PROGRAM EM04_Follower3
VAR
	ref_Master: REFERENCE TO UDT_AXISADMIN;
	ref_Follower: REFERENCE TO UDT_AXISADMIN;
	Ref_MachineStateModel: REFERENCE TO PackMlv3_StateModel;
	Ref_Unit: REFERENCE TO UDT_UnitAdmin;
	EM_No: INT:=4;
	tonAbortingWatchDog: TON;
	tonStoppingWatchDog: Ton;
	MC_CamIn_Follower: MC_CamIn;

	MC_CamTableSelect_Follower: MC_CamTableSelect;
	CamTableFollower: MC_CAM_REF;
	table1: ARRAY[1..2] OF MC_MotionFunctionPoint; (*用于定义电子凸轮表中的关键点*)


    MC_ReadCamTableSlaveDynamicsFollwer: MC_ReadCamTableSlaveDynamics;
	
	tonFollowerSeq: TON;
	FollowerSeq: SequenceTransfer;	
	
	i: INT;
	lrPosCnt: INT;
	bRecipeComplete: BOOL;
	bBeltInRange: BOOL;
	iLastSeq: INT;
END_VAR

VAR CONSTANT
	iCamID: MC_CAM_ID:=3;		
END_VAR

(*减速比10/1 同步轮周长400 ，皮带总长11600，58个工位，工位间距200
28个工位后开始落料*)
Ref_MachineStateModel REF= UN01_MachineStateModel;
Ref_Unit REF=Unit01;
ref_Master REF= arVirtualAxisAdmin[1];
ref_Follower REF= arRealAxisAdmin[43];
MainRoution();
CM01_Cam();
SR999_Faulthandler();

ACTION CM01_Cam:
//凸轮1曲线
camTableFollower.ArraySize:=SIZEOF(table1);
camTableFollower.NoOfColumns:=1;
camTableFollower.NoOfRows:=2;
camTableFollower.pArray:=ADR(table1);
camTableFollower.TableType:=MC_TABLETYPE_MOTIONFUNCTION;

table1[1].FunctionType:=MOTIONFUNCTYPE_POLYNOM1;
table1[1].MasterPos:=0;
table1[1].SlavePos:=0;
table1[1].PointIndex:=1;
table1[1].PointType:=MOTIONPOINTTYPE_MOTION;
		
table1[2].FunctionType:=MOTIONFUNCTYPE_POLYNOM1;
table1[2].MasterPos:=200;
table1[2].SlavePos:=200;
table1[2].PointIndex:=2;
table1[2].PointType:=MOTIONPOINTTYPE_MOTION;

MC_CamIn_Follower(
	Master:= ref_Master.Axis, 
	Slave:= ref_Follower.Axis, 
	Execute:= ref_Follower.i.CamIn , 
	MasterOffset:= , 
	SlaveOffset:= , 
	MasterScaling:= 1, 
	SlaveScaling:= 1, 
	StartMode:= MC_STARTMODE_ABSOLUTE, 
	CamTableID:= iCamID, 
	BufferMode:= , 
	Options:= , 
	InSync=> , 
	Busy=> , 
	Active=> , 
	CommandAborted=> , 
	Error=> , 
	ErrorID=> );
	
MC_CamTableSelect_Follower(
	Master:= ref_Master.Axis, 
	Slave:= ref_Follower.Axis, 
	CamTable:= CamTableFollower, 
	Execute:= ref_Follower.i.SelectCamTable , 
	Periodic:= TRUE, 
	MasterAbsolute:= , 
	SlaveAbsolute:= , 
	CamTableID:= iCamID, 
	Done=> ref_Follower.o.SelectCamTableDone, 
	Busy=> , 
	Error=> , 
	ErrorID=> );	
	
MC_ReadCamTableSlaveDynamicsFollwer(
	Execute:= , 
	CamTableID:=iCamID , 
	MasterPosition:=ref_Master.o.ActPos, 
	Done=> , 
	Busy=> , 
	Error=> , 
	ErrorID=> , 
	SlavePosition=> , 
	SlaveVelocity=> , 
	SlaveAcceleration=> );
END_ACTION

ACTION CM02_Follower:
CASE FollowerSeq.Now OF
	0: 	   
	   IF Ref_MachineStateModel.Sts_Resetting  THEN
          FollowerSeq(ExeCute:=TRUE , Next:= Seq_Resetting);  
	   END_IF	
	
	   IF Ref_MachineStateModel.Sts_Stopping  THEN
		  FollowerSeq(ExeCute:=TRUE , Next:= Seq_Stopping);   
	   END_IF
	   IF Ref_MachineStateModel.Sts_Execute  THEN
		  FollowerSeq(ExeCute:= TRUE, Next:= 110);   
	   END_IF	   
{#region resetting}	   
	Seq_Resetting:
		IF NOT ref_Follower.o.PowerOn  THEN;
		   ref_Follower.i.Enable:=TRUE;
		ELSE
		   FollowerSeq(ExeCute:=TRUE , Next:= 20); 
		END_IF
	    IF Ref_MachineStateModel.Sts_Stopping  THEN
		   FollowerSeq(ExeCute:= TRUE, Next:= Seq_Stopping);  
	    END_IF
		
	20:	
		IF NOT glb_AllAxisHomed_UN01 THEN
			FollowerSeq(ExeCute:=TRUE , Next:= 21);  
			ELSE
			FollowerSeq(ExeCute:=TRUE , Next:= 30); 
		END_IF
	   
	21:
	   iLastSeq:=0;
	   glb_lrBelt3TargetCnt:=0;
	   glb_lrBelt3WrkCnt:=0;
	   glb_lrBelt3ValidCnt:=0;
	   bRecipeComplete:=FALSE;
	   arDropBufferCyclinder[1].i.ActiveIn:=TRUE;
	   arDropBufferCyclinder[1].i.ActiveOut:=FALSE;
	   MEMSET(destAddr:= ADR(glb_BinBelt3), fillByte:= 0, n:= SIZEOF(glb_BinBelt3));      
	   FollowerSeq(ExeCute:=TRUE , Next:= 22); 
	22:
       tonFollowerSeq(IN:=TRUE , PT:=T#1S , Q=> , ET=> );
       IF tonFollowerSeq.Q AND arDropBufferCyclinder[1].I.InSensor 
       AND arDropBufferCyclinder[2].i.InSensor THEN
		   tonFollowerSeq(IN:=FALSE , PT:=T#1S , Q=> , ET=> );
		   FollowerSeq(ExeCute:=TRUE , Next:= 23); 
       END_IF 
	   
	23:
	   ref_Follower.i.Home:=TRUE;
	   IF ref_Follower.o.HomeDone THEN
		   ref_Follower.i.Home:=FALSE;
		   FollowerSeq(ExeCute:=TRUE , Next:= 24); 
	   ELSE IF Ref_MachineStateModel.Sts_Stopping  THEN
		       ref_Follower.i.Home:=FALSE;
			   ref_Follower.i.Stop:=TRUE;
               FollowerSeq(ExeCute:=TRUE , Next:= Seq_Stopping);   
	        END_IF	   
	   END_IF	
		
    24: 
		glb_BinBelt3.bin[1].arDrop[HMI_B3DropBinNo1]:=TRUE;
		glb_BinBelt3.bin[1].arDrop[HMI_B3DropBinNo2]:=TRUE;
		glb_BinBelt3.bin[1].arDrop[HMI_B3DropBinNo3]:=TRUE;
        lrPosCnt:=1;
		ref_Follower.i.Pos:=0;		
		FollowerSeq(ExeCute:=TRUE , Next:= 25);
		
	25:
        IF ref_Follower.o.StandStill THEN
		   FollowerSeq(Execute:= TRUE, Next:= 30);   
	    END_IF
		
    30:	//生产复位
	    ref_Follower.i.MoveAbs:=TRUE; 	
    	IF  ref_Follower.o.CmdDone THEN
		    ref_Follower.i.MoveAbs:=FALSE;
            FollowerSeq(Execute:= TRUE, Next:= Seq_ResettingDone);    	
		END_IF

		
   	Seq_ResettingDone: 
         IF NOT Ref_MachineStateModel.Sts_Resetting THEN
			FollowerSeq(ExeCute:=TRUE , Next:= 0); 	
		 END_IF	   
{end_region}
	
    //自动运行
    110:
        IF iLastSeq>100 THEN
	       FollowerSeq(ExeCute:=TRUE , Next:= iLastSeq);
        ELSE 
		   FollowerSeq(ExeCute:=TRUE , Next:= 111);
		END_IF
    111: 
        IF glb_BinBelt1.bin[HMI_B1DropBinNo].arDrop[HMI_B1DropBinNo] THEN //等待皮带1倒药
		   FollowerSeq(ExeCute:=TRUE , Next:= 112);
		END_IF
		
		IF NOT glb_BinBelt1.bin[HMI_B1DropBinNo].arDrop[HMI_B1DropBinNo] 
		   AND glb_lrBelt3ValidCnt > 0  THEN // AND glb_lrBelt1WrkCnt=0 
			FollowerSeq(ExeCute:=TRUE , Next:= 120);
		END_IF
		
		IF Ref_MachineStateModel.Sts_Stopping  THEN
			FollowerSeq(ExeCute:=TRUE , Next:= Seq_Stopping);   
		END_IF   		
    112:
		   glb_BinBelt3.bin[1].arDrop[HMI_B3DropBinNo1]:=TRUE;
//		   glb_BinBelt3.bin[1].arDrop[HMI_B3DropBinNo2]:=FALSE;
//		   glb_BinBelt3.bin[1].arDrop[HMI_B3DropBinNo3]:=FALSE; 
           FollowerSeq(ExeCute:=TRUE , Next:= 120); 	
    120:  
	      IF NOT glb_BinBelt3.bin[HMI_B3DropBinNo1].arDrop[HMI_B3DropBinNo1] 
          AND NOT glb_BinBelt3.bin[HMI_B3DropBinNo2].arDrop[HMI_B3DropBinNo2] THEN 
              FollowerSeq(ExeCute:=TRUE , Next:= 121); 	
		  END_IF
		  IF Ref_MachineStateModel.Sts_Stopping  THEN
		     FollowerSeq(ExeCute:=TRUE , Next:= Seq_Stopping);   
	      END_IF
		  
    121: 
         IF NOT glb_BinBelt3.bin[HMI_B3DropBinNo3].arDrop[HMI_B3DropBinNo3] THEN
             FollowerSeq(ExeCute:=TRUE , Next:= 130); 	
	     ELSE 
		     FollowerSeq(ExeCute:=TRUE , Next:= 200); //往皮带4倒药	
         END_IF
	130:  
	      ref_Follower.i.Pos:=ref_Follower.i.Pos+200;
	      FollowerSeq(ExeCute:=TRUE ,Hold:=FALSE, Next:= 150);
	
	150:
	      ref_Follower.i.MoveAbs:=TRUE;
		  IF ref_Follower.o.CmdDone THEN
			 ref_Follower.i.MoveAbs:=FALSE;
			 FollowerSeq(ExeCute:=TRUE ,Hold:=FALSE, Next:= 300);
		  END_IF
	
	//往皮带4落料
	200:
	     IF glb_BinBelt4_5.bin[1].arDrop[1] THEN
			FollowerSeq(ExeCute:=TRUE , Next:= 210); 
		 END_IF
		 IF Ref_MachineStateModel.Sts_Stopping  THEN
		    FollowerSeq(ExeCute:=TRUE , Next:= Seq_Stopping);   
	     END_IF
	
	210:
		ref_Follower.i.Pos:=ref_Follower.i.Pos+200;
		FollowerSeq(ExeCute:=TRUE ,Hold:=FALSE, Next:= 220);
	
	220:
	      ref_Follower.i.MoveAbs:=TRUE;
		  IF ref_Follower.o.CmdDone THEN
			 ref_Follower.i.MoveAbs:=FALSE;
			 FollowerSeq(ExeCute:=TRUE ,Hold:=FALSE, Next:= 230);
		  END_IF	
		  IF (ref_Follower.i.Pos-ref_Follower.o.ActPos) < 60 AND NOT bBeltInRange THEN
				glb_BinBelt4_5.bin[1].arDrop[1]:=FALSE;
				glb_BinBelt4_5.bin[1].Name:= glb_BinBelt3.bin[HMI_B3DropBinNo3].Name;
				glb_BinBelt4_5.bin[1].Amount:= glb_BinBelt3.bin[HMI_B3DropBinNo3].Amount;
				glb_BinBelt4_5.bin[1].bReject:= glb_BinBelt3.bin[HMI_B3DropBinNo3].bReject;
				glb_lrBelt3ValidCnt:=glb_lrBelt3ValidCnt-1;
			  bBeltInRange:=TRUE;
		  END_IF 
	
	230:  
	      bBeltInRange:=FALSE;
		  glb_BinBelt3.bin[HMI_B3DropBinNo3].arDrop[HMI_B3DropBinNo3]:=FALSE;
		  FollowerSeq(ExeCute:=TRUE ,Hold:=FALSE, Next:= 300); 
		  
    300: 
	
			FOR i:=64 TO 1 BY -1 DO
				glb_BinBelt3.bin[i]:= glb_BinBelt3.bin[i-1];  
			END_FOR	     
			glb_BinBelt3.bin[1].arDrop[HMI_B3DropBinNo1]:=FALSE;
			glb_BinBelt3.bin[1].arDrop[HMI_B3DropBinNo2]:=FALSE;
			glb_BinBelt3.bin[1].arDrop[HMI_B3DropBinNo3]:=FALSE;
			glb_lrBelt3WrkCnt:=glb_lrBelt3WrkCnt+1;
			FollowerSeq(ExeCute:=TRUE ,Hold:=FALSE, Next:= 111);  

			
		  
	Seq_Stopping: 
        iLastSeq:= FollowerSeq.Last; 
	    tonFollowerSeq(IN:=TRUE , PT:=T#1S , Q=> , ET=> );
		IF tonFollowerSeq.Q THEN
			tonFollowerSeq(IN:=FALSE , PT:=T#1S , Q=> , ET=> );
			FollowerSeq(ExeCute:=TRUE , Next:= Seq_StoppingDone); 
		END_IF
		
	Seq_StoppingDone:
	     ref_Follower.i.Disable:=TRUE;
		 IF NOT Ref_MachineStateModel.Sts_Stopping THEN
			FollowerSeq(ExeCute:=TRUE , Next:= 0); 
		 END_IF
END_CASE
FollowerSeq.Hold := Ref_MachineStateModel.Sts_Held;
END_ACTION

ACTION MainRoution:
EM_No:=4;
IF Ref_Unit.EM_Selected[EM_No] THEN
	IF Ref_MachineStateModel.Sts_Holding THEN
		Ref_Unit.EM_Holding_Done[EM_No]:=TRUE;
		ELSE
		Ref_Unit.EM_Holding_Done[EM_No]:=FALSE;
	END_IF
	IF Ref_MachineStateModel.Sts_UnHolding THEN
		Ref_Unit.EM_UnHolding_Done[EM_No]:=TRUE;
		ELSE
		Ref_Unit.EM_UnHolding_Done[EM_No]:=FALSE;
	END_IF
	
	IF Ref_MachineStateModel.Sts_Suspending THEN
		Ref_Unit.EM_Suspending_Done[EM_No]:=TRUE;
		ELSE
		Ref_Unit.EM_Suspending_Done[EM_No]:=FALSE;
	END_IF
	
	IF Ref_MachineStateModel.Sts_UnSuspending THEN
		Ref_Unit.EM_UnSuspending_Done[EM_No]:=TRUE;
		ELSE
		Ref_Unit.EM_UnSuspending_Done[EM_No]:=FALSE;
	END_IF
	
	IF Ref_MachineStateModel.Sts_Resetting AND FollowerSeq.Now=Seq_ResettingDone THEN
	   Ref_Unit.EM_Resetting_Done[EM_No]:=TRUE;
       ELSE   
	   Ref_Unit.EM_Resetting_Done[EM_No]:=FALSE;
	END_IF
	
	IF Ref_MachineStateModel.Sts_Clearing THEN
	   Ref_Unit.EM_Clearing_Done[EM_No]:=TRUE;
	   ELSE
	   Ref_Unit.EM_Clearing_Done[EM_No]:=FALSE;
	END_IF
	
	IF Ref_MachineStateModel.Sts_Starting THEN
	   Ref_Unit.EM_Starting_Done[EM_No]:=TRUE;
	   ELSE
       Ref_Unit.EM_Starting_Done[EM_No]:=FALSE;
	END_IF
	
	IF Ref_MachineStateModel.Sts_Stopping AND FollowerSeq.Now=Seq_StoppingDone  THEN
	   Ref_Unit.EM_Stopping_Done[EM_No]:=TRUE;	
       ELSE  
	   Ref_Unit.EM_Stopping_Done[EM_No]:=FALSE;	
	END_IF

	IF Ref_MachineStateModel.Sts_Aborting THEN
	    FollowerSeq(ExeCute:=TRUE , Next:= 0);	
		IF ref_Follower.o.InSync THEN	 
		   ref_Follower.i.CamOut:=TRUE;
		ELSE IF  NOT ref_Follower.o.StandStill THEN
				ref_follower.i.Stop:=TRUE;
			END_IF
		END_IF  
		
		IF tonAbortingWatchDog.Q THEN 
			Ref_Unit.EM_Aborting_Done[EM_No]:=TRUE;
			ref_Follower.i.Disable:=TRUE;
        END_IF
    ELSE
		Ref_Unit.EM_Aborting_Done[EM_No]:=FALSE;
	END_IF
	
	tonAbortingWatchDog(IN:= Ref_MachineStateModel.Sts_Aborting, PT:=T#3S , Q=> , ET=> );
	CM02_Follower();
ELSE
FollowerSeq(ExeCute:=TRUE , Next:= 0); 			
END_IF
END_ACTION

ACTION SR999_FaultHandler:
;
END_ACTION

END_PROGRAM

(* stored: Version 1.1.0.1, ProductVersion 3.1.4024.6
   POU EM04_Follower3: Id {649c12a4-874d-4d73-8db5-fadb49cbf83a}, SpecialFunc None
   Action CM01_Cam: Id {72b77851-d151-48c8-8aa3-67f6cd68a1dc}
   Action CM02_Follower: Id {a4b9b18c-3c32-48f7-ae49-cb984ac32f7f}
   Action MainRoution: Id {45c00345-45dd-4368-8aeb-216ef3a4244b}
   Action SR999_FaultHandler: Id {e1a75517-513f-479f-a1a4-c8f363ed63c7} *)
